# EPICS substitutions: ek9000App/Db/EL1104.substitutions
file EL1104.template
{ 	pattern
	{
		TERMINAL,

	}
	{
	}
}
